Staubli VAL3: ReadMe.pgx

program ReadMe()
begin
//在通用版本上对lasman进行定制
//1.添加了三个四个函数
//checkAxis
//SingleMove
//RecordExtAxis
//RecordJoint


//还有一些变量需要添加







end
